// TIA Portal V17 export
// export: Created 2022-07-20T07:01:27.0002203Z, ExportSetting WithDefaults, DisplayName Totally Integrated Automation Portal, DisplayVersion V17, DisplayName TIA Portal Openness, DisplayVersion V17, DisplayName TIA Portal Version Control Interface, DisplayVersion V17, DisplayName SINAMICS Startdrive Advanced, DisplayVersion V17, DisplayName SINAMICS Startdrive G130, G150, S120, S150, SINAMICS MV, S210, DisplayVersion V17, DisplayName SINAMICS Startdrive G110M, G120, G120C, G120D, G120P, G115D, DisplayVersion V17, DisplayName STEP 7 Professional, DisplayVersion V17, DisplayName STEP 7 Safety, DisplayVersion V17, DisplayName WinCC Advanced, DisplayVersion V17
FUNCTION_BLOCK "FB10030_AnalogicalSensor"   // FB10030, LAD
{ S7_Optimized_Access := 'TRUE' }
VERSION : 0.1
// stored: AutoNumber false, IsIECCheckEnabled false, IsRetainMemResEnabled false, MemoryReserve 100, SetENOAutomatically false, UDAEnableTagReadback false
   VAR_INPUT
      RawValue : Int;
      CalibrationValue_1 : Real;
      CalibrationValue_2 : Real;
      Unit : SInt;   // 0 = Calibration Value Unit, 1 = %
      ReverseScale : Bool;
      HighErrorThreshold : Real;
      HighWarningThreshold : Real;
      LowWarningThreshold : Real;
      LowErrorThreshold : Real;
   END_VAR
   VAR_OUTPUT
      SensorCalibrated : Bool;
      CalibrationStatus_1 : Bool;
      CalibrationStatus_2 : Bool;
      ActualValue : Real;   // Depend On The Calibration Value
      "ActualValue_%" : Real;
      HighErrorThresholdReached : Bool;
      HighWarningThresholdReached : Bool;
      LowWarningThresholdReached : Bool;
      LowErrorThresholdReached : Bool;
   END_VAR
   VAR_IN_OUT
      RequestCalibration_1 : Bool;
      RequestResetCalibration : Bool;
      RequestCalibration_2 : Bool;
      CalibrationDataX_1 : Real;
      CalibrationDataY_1 : Real;   // mm
      CalibrationDataX_2 : Real;
      CalibrationDataY_2 : Real;   // mm
   END_VAR
BEGIN

REGION Network 1 (SCL): Sensor Calibration Management
   //Calibration 1 Management
   IF #RequestCalibration_1 THEN
       #CalibrationDataX_1 := #RawValue;
       #CalibrationDataY_1 := #CalibrationValue_1;
       #CalibrationStatus_1 := TRUE;
       #RequestCalibration_1 := FALSE;
   END_IF;

   //Calibration 2 Management
   IF #RequestCalibration_2 THEN
       #CalibrationDataX_2 := #RawValue;
       #CalibrationDataY_2 := #CalibrationValue_2;
       #CalibrationStatus_2 := TRUE;
       #RequestCalibration_2 := FALSE;
   END_IF;

   //Reset Calibration Management
   IF #RequestResetCalibration THEN
       #CalibrationDataX_1 := 0;
       #CalibrationDataY_1 := 0;
       #CalibrationStatus_1 := FALSE;
       #CalibrationDataX_2 := 0;
       #CalibrationDataY_2 := 0;
       #CalibrationStatus_2 := FALSE;
       #RequestResetCalibration := FALSE;
   END_IF;
END_REGION

REGION Network 2 (SCL): Process Value Management
   IF #SensorCalibrated THEN
       //Determine The Process Value By Linearization
       IF NOT(#ReverseScale) THEN
           "FC10020_Linearization"(X1 := #CalibrationDataX_1,
                                   Y1 := #CalibrationDataY_1,
                                   X2 := #CalibrationDataX_2,
                                   Y2 := #CalibrationDataY_2,
                                   X := #RawValue,
                                   Y => #ActualValue);
       ELSE
           "FC10020_Linearization"(X1 := #CalibrationDataX_1,
                                   Y1 := #CalibrationDataY_1,
                                   X2 := #CalibrationDataX_2,
                                   Y2 := #CalibrationDataY_2,
                                   X := #RawValue,
                                   Y => #ActualValue);
           #ActualValue := #CalibrationDataY_2 - #ActualValue;
       END_IF;


       //Determine the distance in percentage
       IF #CalibrationDataY_2 <> 0 THEN
           #"ActualValue_%" := (#ActualValue * 100) / #CalibrationDataY_2;
       ELSE
           #"ActualValue_%" := 0.0;
       END_IF;
   ELSE
       #ActualValue := #RawValue;
   END_IF;
END_REGION

REGION Network 3 (SCL): Sensor States Management
   //Sensor Calibrated Management
   IF
       ((#CalibrationDataX_1 = #CalibrationDataY_1) AND (#CalibrationDataY_1 = #CalibrationDataX_2) AND (#CalibrationDataX_2  = #CalibrationDataY_2) AND (#CalibrationDataY_2 = 0)) OR
       (#CalibrationDataX_1 = #CalibrationDataX_2) OR
       (#CalibrationDataY_1 = #CalibrationDataY_2)
   THEN
       #SensorCalibrated := FALSE;
   ELSE
       #SensorCalibrated := TRUE;
   END_IF;

   //Thresholds Management
   IF #SensorCalibrated THEN
       IF ((#Unit = 0 AND #ActualValue > #HighErrorThreshold) OR (#Unit = 1 AND #"ActualValue_%" > #HighErrorThreshold)) THEN
           #HighErrorThresholdReached := TRUE;
       ELSE
           #HighErrorThresholdReached := FALSE;
       END_IF;

       IF ((#Unit = 0 AND #ActualValue > #HighWarningThreshold) OR (#Unit = 1 AND #"ActualValue_%" > #HighWarningThreshold)) THEN
           #HighWarningThresholdReached := TRUE;
       ELSE
           #HighWarningThresholdReached := FALSE;
       END_IF;

       IF ((#Unit = 0 AND #ActualValue < #LowWarningThreshold) OR (#Unit = 1 AND #"ActualValue_%" < #LowWarningThreshold)) THEN
           #LowWarningThresholdReached := TRUE;
       ELSE
           #LowWarningThresholdReached := FALSE;
       END_IF;

       IF ((#Unit = 0 AND #ActualValue < #LowErrorThreshold) OR (#Unit = 1 AND #"ActualValue_%" < #LowErrorThreshold)) THEN
           #LowErrorThresholdReached := TRUE;
       ELSE
           #LowErrorThresholdReached := FALSE; 
       END_IF;
   ELSE
       #HighErrorThresholdReached := TRUE;
       #HighWarningThresholdReached := TRUE;
       #LowWarningThresholdReached := TRUE;
       #LowErrorThresholdReached := TRUE;
   END_IF;
END_REGION
END_FUNCTION_BLOCK
